DATA_BLOCK "dbParTank"
{ S7_Optimized_Access := 'TRUE' }
VERSION : 0.8
NON_RETAIN
   VAR
      parTank { ExternalAccessible := 'False'; ExternalVisible := 'False'; ExternalWritable := 'False'} : Array[1..25] of "tParameterTank";
      ia { ExternalAccessible := 'False'; ExternalVisible := 'False'; ExternalWritable := 'False'} : "tIndex";
      firstRunning { ExternalAccessible := 'False'; ExternalVisible := 'False'; ExternalWritable := 'False'} : "tStatus";
   END_VAR


BEGIN

END_DATA_BLOCK

